FUNCTION alg_g_z2: LREAL
VAR_INPUT
    state: STATE;
END_VAR

alg_g_z2 := state.curTime;

END_FUNCTION

(* stored: ProductVersion 3.1.0.18, Version 1.1.0.1 *)
